// Status of FB_DigitalInput. `header` is shared with every other device FB
// (see ST_DeviceHeader_Sts); device-specific fields sit below.
{attribute 'OPC.UA.DA' := '1'}
{attribute 'OPC.UA.DA.Access' := '1'}
{attribute 'OPC.UA.DA.StructuredType' := '1'}
TYPE ST_DigitalInput_Sts :
STRUCT
    header        : ST_DeviceHeader_Sts;

    {attribute 'OPC.UA.DA.Description' := 'Final processed value (after invert + debounce)'}
    value      : BOOL;
    {attribute 'OPC.UA.DA.Description' := 'Raw terminal reading (before invert / debounce)'}
    rawValue   : BOOL;
    {attribute 'OPC.UA.DA.Description' := 'Signal quality tag'}
    quality    : E_IO_Quality := E_IO_Quality.UNKNOWN;
    {attribute 'OPC.UA.DA.Description' := 'One-scan pulse on debounced rising edge'}
    risingEdge : BOOL;
    {attribute 'OPC.UA.DA.Description' := 'One-scan pulse on debounced falling edge'}
    fallingEdge: BOOL;
END_STRUCT
END_TYPE

(* stored: Version 1.1.0.1, ProductVersion 3.1.4026.12
   DUT ST_DigitalInput_Sts: Id {b0100001-0002-0000-0000-000000000001} *)
